// TIA Portal V16 export
// export: Created 2021-11-12T13:33:05.2761645Z, ExportSetting WithDefaults, DisplayName Totally Integrated Automation Portal, DisplayVersion V16 Update 3, DisplayName TIA Portal Version Control Interface, DisplayVersion V16 Update 2, DisplayName TIA Portal Openness, DisplayVersion V16 Update 3, DisplayName SINAMICS Startdrive Advanced, DisplayVersion V16 Update 5, DisplayName SINAMICS Startdrive G130, G150, S120, S150, SINAMICS MV, S210, DisplayVersion V16 Update 5, DisplayName SINAMICS Startdrive G110M, G120, G120C, G120D, G120P, G115D, DisplayVersion V16 Update 5, DisplayName STEP 7 Professional, DisplayVersion V16 Update 3, DisplayName STEP 7 Safety, DisplayVersion V16, DisplayName WinCC UA Professional, DisplayVersion V16 Update 3
DATA_BLOCK "HMI_PARAM_460"   // DB106
{ S7_Optimized_Access := 'TRUE' }
VERSION : 0.1
// stored: AutoNumber true, DBAccessibleFromOPCUA true, IsOnlyStoredInLoadMemory false, IsRetainMemResEnabled false, IsWriteProtectedInAS false, MemoryReserve 100
   VAR
      xxxxx___BinarySensors___xxxxx : Byte;
      "GL01-BG01" : "UDT_CH_DI_Parameter";   // Reflexní optická závora - Snímání pohybu dílu na dopravníku
      "GL02-BG01" : "UDT_CH_DI_Parameter";   // Reflexní optická závora - Snímání pohybu dílu na dopravníku
      "GL03-BG01" : "UDT_CH_DI_Parameter";   // Reflexní optická závora - Snímání pohybu dílu na dopravníku
      "GL04-BG01" : "UDT_CH_DI_Parameter";   // Reflexní optická závora - Snímání pohybu dílu na dopravníku
      "UC21-FC01_14" : "UDT_CH_DI_Parameter";   // 400V Dopravník ++460 OK
      "UC21-FC02_14" : "UDT_CH_DI_Parameter";   // 400V Dopravník ++460 OK
      "UC21-FC03_14" : "UDT_CH_DI_Parameter";   // 400V Dopravník ++460 OK
      "UC21-FC04_14" : "UDT_CH_DI_Parameter";   // 400V Dopravník ++460 OK
      "GL01-BG01_4" : "UDT_CH_DI_Parameter";   // Snímání pohybu dílu na dopravníku ++460+GL01 (M1)
      "GL02-BG01_4" : "UDT_CH_DI_Parameter";   // Snímání pohybu dílu na dopravníku ++460+GL02 (M3)
      "GL03-BG01_4" : "UDT_CH_DI_Parameter";   // Snímání pohybu dílu na dopravníku ++460+GL03 (M7.2)
      "GL04-BG01_4" : "UDT_CH_DI_Parameter";   // Snímání pohybu dílu na dopravníku ++460+GL04 (M5)
      xxxxx___BinaryOthers___xxxxx : Byte;
      "UH11-SF01_14" : "UDT_CH_DI_Parameter";   // Conveyor Remote
      "UH11-SF01_24" : "UDT_CH_DI_Parameter";   // Conveyor Automat
      "UH11-SF03_14" : "UDT_CH_DI_Parameter";   // Conveyor Start automat
      "UH11-SF04_12" : "UDT_CH_DI_Parameter";   // Conveyor Stop
      "UH11-SF05_14" : "UDT_CH_DI_Parameter";   // Conveyor GL02 Manual Backward
      "UH11-SF05_24" : "UDT_CH_DI_Parameter";   // Conveyor GL02 Manual Forward
      "UH11-SF06_14" : "UDT_CH_DI_Parameter";   // Conveyor GL03 Manual Backward
      "UH11-SF06_24" : "UDT_CH_DI_Parameter";   // Conveyor GL03 Manual Forward
      "UH11-SF07_14" : "UDT_CH_DI_Parameter";   // Conveyor GL04 Manual Backward
      "UH11-SF07_24" : "UDT_CH_DI_Parameter";   // Conveyor GL04 Manual Forward
      "UH11-SF08_14" : "UDT_CH_DI_Parameter";   // Bedna Žádost o výměnu
      "UH11-SF09_14" : "UDT_CH_DI_Parameter";   // Bedna vyměněna
      "UH31-SF07_14" : "UDT_CH_DI_Parameter";   // Conveyor GL01 Remote
      UH31_SF07_24 : "UDT_CH_DI_Parameter";   // Conveyor GL01 Automat
      "UH31-SF09_14" : "UDT_CH_DI_Parameter";   // Conveyor GL01 Start automat
      "UH31-SF10_12" : "UDT_CH_DI_Parameter";   // Conveyor GL01 Stop
      "UH31-SF08_14" : "UDT_CH_DI_Parameter";   // Conveyor GL01 Manual Backward
      "UH31-SF08_24" : "UDT_CH_DI_Parameter";   // Conveyor GL01 Manual Forward
      "UH31-SF11_X2" : "UDT_CH_DI_Parameter";   // Dopravník GL01 - blokování pásu v kleci
      xxxxx___Drives___xxxxx : Byte;
      "GL01-MA01" : "UDT_Drive1_Parameter";   // Dopravník ke tryskači (M1)
      "GL02-MA01" : "UDT_Drive1_Parameter";   // Dopravník ke tryskači (M3)
      "GL03-MA01" : "UDT_Drive1_Parameter";   // Dopravník ke tryskači (M7.2)
      "GL04-MA01" : "UDT_Drive1_Parameter";   // Dopravník ke tryskači (M5)
      "UC21-TA01" : "UDT_SINAMICS_G120_Parameter";   // Měnič
      "UC21-TA02" : "UDT_SINAMICS_G120_Parameter";   // Měnič
      "UC21-TA03" : "UDT_SINAMICS_G120_Parameter";   // Měnič
      "UC21-TA04" : "UDT_SINAMICS_G120_Parameter";   // Měnič
      xxxxx___Others___xxxxx : Byte;
      CL01 : "UDT_PartCounter_Parameter";   // Box
   END_VAR
   VAR RETAIN
      TOFTime_440TA01_PT : Time := T#60s;   // TOF time to stop conv after 440TA01 stopped
      TOFTime_460TA01_PT : Time := T#60s;   // TOF time to stop conv after 460TA01 stopped
      TOFTime_460TA02_1_PT : Time := T#60s;   // TOF time to stop conv after 460TA02 stopped
      TOFTime_460TA02_2_PT : Time := T#60s;   // TOF time to stop conv after 460TA02 stopped
   END_VAR
   VAR
      TOFTime_460TA04_PT : Time := T#60s;   // TOF time to stop conv after 460TA03 stopped
      xxxxx___Alarms___xxxxx : Byte;
      CL01_Alarm : "UDT_DI_Mon_Parameter";   // CL01 - box full
      CL01_Warn : "UDT_DI_Mon_Parameter";   // CL01 - box full
   END_VAR
BEGIN
   "UC21-TA01".RefSpdP2000 := 1500.0;
   "UC21-TA01".RefCurrP2002 := 2.49;
   "UC21-TA01".RefTrqP2003 := 7.29;
   "UC21-TA02".RefSpdP2000 := 1500.0;
   "UC21-TA02".RefCurrP2002 := 2.49;
   "UC21-TA02".RefTrqP2003 := 7.29;
   "UC21-TA03".RefSpdP2000 := 1500.0;
   "UC21-TA03".RefCurrP2002 := 2.49;
   "UC21-TA03".RefTrqP2003 := 7.29;
   "UC21-TA04".RefSpdP2000 := 1500.0;
   "UC21-TA04".RefCurrP2002 := 2.49;
   "UC21-TA04".RefTrqP2003 := 7.29;
   CL01_Warn.Func := 16#2;
END_DATA_BLOCK
